# EPICS autosave request: tests/testfiles/cfg/SF_OpticsMQUA_PV.req
$(SYS):ONOFF
$(SYS):K1L-SET
